// TIA Portal V17 export
// export: Created 2024-09-02T12:50:26.7070187Z, ExportSetting WithDefaults, DisplayName Totally Integrated Automation Portal, DisplayVersion V17, DisplayName TIA Portal Openness, DisplayVersion V17, DisplayName TIA Portal Version Control Interface, DisplayVersion V17, DisplayName STEP 7 Professional, DisplayVersion V17, DisplayName STEP 7 Safety, DisplayVersion V17, DisplayName WinCC Professional, DisplayVersion V17
TYPE "TypeOperatingModesHMI"
// stored: IsFailsafeCompliant false
   STRUCT
      Buttons : Struct
         Active : Bool;
         MediaON : Bool;
         MediaOFF : Bool;
         Hand : Bool;
         Auto : Bool;
         StartOn : Bool;
         StartOff : Bool;
         TactEnd : Bool;
         Home : Bool;
      END_STRUCT;
      RM : Struct
         Active : Bool;
         MediaON : Bool;
         MediaOFF : Bool;
         Hand : Bool;
         Auto : Bool;
         StartOn : Bool;
         StartOff : Bool;
         TactEnd : Bool;
         Home : Bool;
      END_STRUCT;
   END_STRUCT;
END_TYPE
